FUNCTION TryConvert_LINT_TO_DT : BOOL
VAR_INPUT
	in : LINT;
	out : REFERENCE TO DT;
END_VAR

IF in > DatatypeLimits.MAX_VALUE_OF_LINT_WHICH_CAN_BE_HELD_IN_A_DT THEN
	RETURN;
END_IF

IF in < DatatypeLimits.MIN_VALUE_OF_LINT_WHICH_CAN_BE_HELD_IN_A_DT THEN
	RETURN;
END_IF

out := LINT_TO_DT(in);
TryConvert_LINT_TO_DT := TRUE;

END_FUNCTION

(* stored: Version 1.1.0.1, ProductVersion 3.1.4024.12
   POU TryConvert_LINT_TO_DT: Id {bfc654c8-9743-4dea-9960-74d84a4d14f0}, SpecialFunc None *)
